{attribute 'linkalways'} 
{attribute 'no_explicit_call' := 'This FB is a CLASS and must be accessed using methods or properties'}
{attribute 'enable_dynamic_creation'}
FUNCTION_BLOCK _ETcVnCalibrationPattern EXTENDS EnumDatatypeBase
VAR
	localData : ETcVnCalibrationPattern;
	activeData : REFERENCE TO ETcVnCalibrationPattern;
	enumBaseDatatype : _DINT(localData);
END_VAR

METHOD PRIVATE AddLocalEnumeration
VAR_INPUT
	Enumeration : T_MAXSTRING;
	Value : ETcVnCalibrationPattern;
END_VAR
AddEnumeration(Enumeration, Value);
END_METHOD

PROPERTY PUBLIC Address : PVOID
GET
Address := ADR(activeData);
END_GET
END_PROPERTY

METHOD PUBLIC ClearReference
VAR_INPUT
END_VAR
activeData REF= localData;
SetBaseDatatypeReference();
END_METHOD

METHOD PUBLIC Clone : I_Datatype
VAR
    pClone : POINTER TO _ETcVnCalibrationPattern;
END_VAR
pClone := __NEW(_ETcVnCalibrationPattern(InitialValue := Value));
Clone := pClone^;
END_METHOD

METHOD FB_init : BOOL
VAR_INPUT
	bInitRetains : BOOL; // if TRUE, the retain variables are initialized (warm start / cold start)
	bInCopyCode : BOOL;  // if TRUE, the instance afterwards gets moved into the copy code (online change)
	InitialValue : ETcVnCalibrationPattern;
END_VAR
localData := InitialValue;
AddBaseDatatype(enumBaseDatatype);
ClearReference();

AddLocalEnumeration('TCVN_CP_CIRCLES_SYM', ETcVnCalibrationPattern.TCVN_CP_CIRCLES_SYM);
AddLocalEnumeration('TCVN_CP_CIRCLES_ASYM', ETcVnCalibrationPattern.TCVN_CP_CIRCLES_ASYM);
AddLocalEnumeration('TCVN_CP_CIRCLES_ASYM_INDENT', ETcVnCalibrationPattern.TCVN_CP_CIRCLES_ASYM_INDENT);
END_METHOD

PROPERTY PUBLIC Identifier : T_MAXSTRING
GET
Identifier := 'ETcVnCalibrationPattern';
END_GET
END_PROPERTY

METHOD IsEnumeratorValueEqual : BOOL
VAR_INPUT
	Enumerator : I_KeyValueForwardEnumerator;
END_VAR
VAR
	storedValue : ETcVnCalibrationPattern;
END_VAR
IF NOT Enumerator.TryGet(storedValue) THEN
	RETURN;
END_IF

IsEnumeratorValueEqual := storedValue = activeData;
END_METHOD

METHOD PUBLIC MakeReferenceTo
VAR_INPUT
	ReferenceTarget : REFERENCE TO ETcVnCalibrationPattern;
END_VAR
activeData REF= ReferenceTarget;
SetBaseDatatypeReference();
END_METHOD

METHOD PROTECTED SetBaseDatatypeReference
VAR_INPUT
END_VAR
enumBaseDatatype.MakeReferenceTo(activeData);
END_METHOD

PROPERTY PUBLIC Size : UDINT
GET
Size := SIZEOF(activeData);
END_GET
END_PROPERTY

METHOD TryMakeReferenceTo : BOOL
VAR_INPUT
	Target : I_Datatype;
END_VAR
VAR
	targetAsEnum : I_EnumDatatype;
	pTargetData : POINTER TO ETcVnCalibrationPattern;
END_VAR
IF NOT Target.TryResolveAsEnumDatatype(targetAsEnum) THEN
	RETURN;
END_IF

IF targetAsEnum.Identifier <> Identifier THEN
	RETURN;
END_IF

pTargetData := Target.Address;
activeData REF= pTargetData^;
SetBaseDatatypeReference();
TryMakeReferenceTo := TRUE;
END_METHOD

PROPERTY PUBLIC Value : ETcVnCalibrationPattern
GET
Value := activeData;
END_GET
SET
activeData := Value;
END_SET
END_PROPERTY

END_FUNCTION_BLOCK

(* stored: Version 1.1.0.1
   POU _ETcVnCalibrationPattern: Id {9f284fa6-0c71-049d-2a70-9bc51a78b1b2}, SpecialFunc None
   Folder Constructor: Id {be28ce50-3b09-0ae5-074e-a72962018730}
   Folder Private: Id {2ddba11a-3bba-04da-37fd-ecefd8d9123d}
   Folder Protected: Id {725fc9ed-3da3-0df9-3517-69a01ff1ddda}
   Method AddLocalEnumeration: Id {9c7b79eb-884b-0c77-2c7a-32401cb96ed4}
   Property Address: Id {223bfad0-4a3d-099d-3131-9156acb18b3e}
   Get Get: Id {930a4d12-7e66-0348-1527-43bc80605b8a}
   Method ClearReference: Id {2ce2e41a-77d6-0c18-0616-2817b0b96ea0}
   Method Clone: Id {0b695f93-906e-089e-1d50-66202890d849}
   Method FB_init: Id {fadd9d0d-3fb9-0032-0f2f-d09a7f2a862c}
   Property Identifier: Id {746fdeb5-9c87-063a-3ddc-d95ff9b8f9c4}
   Get Get: Id {6d348958-787e-0ec6-0c19-bc37f0fb2977}
   Method IsEnumeratorValueEqual: Id {8dc7ab8d-a016-01f2-053f-aead9441d7ec}
   Method MakeReferenceTo: Id {4e042082-937f-0a01-2357-f3fb144bad27}
   Method SetBaseDatatypeReference: Id {d8835c34-6770-0918-3916-d6070ee2baef}
   Property Size: Id {f4e7d02b-fc93-0445-0463-a278815ab256}
   Get Get: Id {e463a6a5-facd-0eaf-08d1-918eb447397a}
   Method TryMakeReferenceTo: Id {34f935dd-1363-03ac-2c70-e125ab08fb19}
   Property Value: Id {294165b5-44b8-08bf-0807-c8f0e8ff5704}
   Get Get: Id {06e6cbd3-74b5-0522-0866-b2f22728f3c9}
   Set Set: Id {4ca6a465-e672-0928-333e-ac0ec7f6b5fc} *)
